TYPE ST_PersistentData_03 :
STRUCT
END_STRUCT
END_TYPE

(* stored: Version 1.1.0.1, ProductVersion 3.1.4024.6
   DUT ST_PersistentData_03: Id {f39d34c5-82ef-4c2a-86b7-156410e422f8} *)
